// Mitsubishi GX Works2 project: 모터실린더완성2   PLC: Q02/Q02H

PROGRAM MAIN
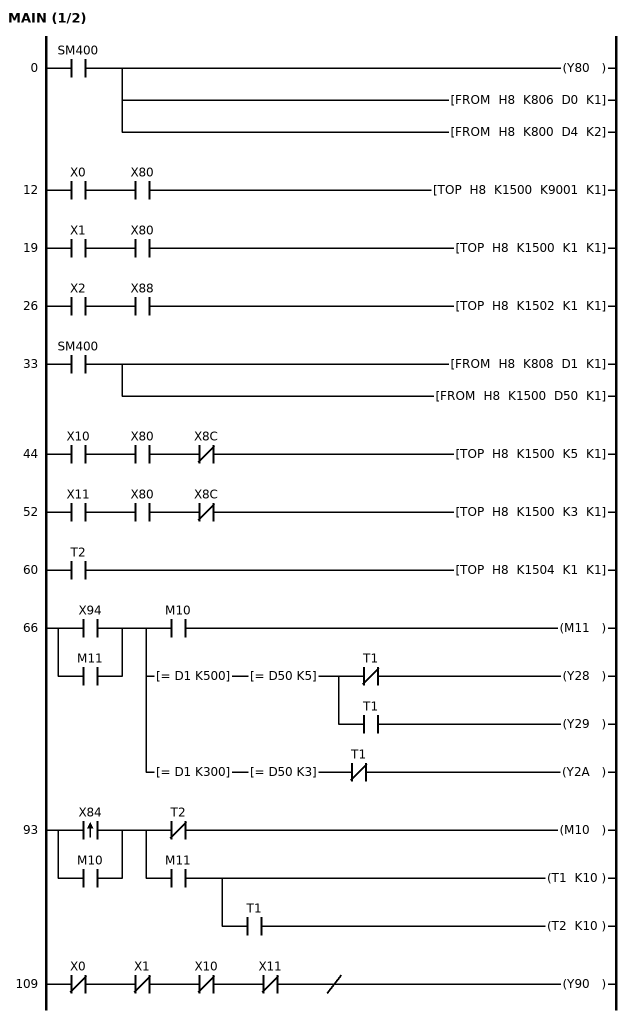
0     LD      SM400
      OUT     Y80
      FROM    H8 K806 D0 K1
      FROM    H8 K800 D4 K2
12    LD      X0
      AND     X80
      TOP     H8 K1500 K9001 K1
19    LD      X1
      AND     X80
      TOP     H8 K1500 K1 K1
26    LD      X2
      AND     X88
      TOP     H8 K1502 K1 K1
33    LD      SM400
      FROM    H8 K808 D1 K1
      FROM    H8 K1500 D50 K1
44    LD      X10
      AND     X80
      ANI     X8C
      TOP     H8 K1500 K5 K1
52    LD      X11
      AND     X80
      ANI     X8C
      TOP     H8 K1500 K3 K1
60    LD      T2
      TOP     H8 K1504 K1 K1
66    LD      X94
      OR      M11
      MPS
      AND     M10
      OUT     M11
      MRD
      AND=    D1 K500
      AND=    D50 K5
      MPS
      ANI     T1
      OUT     Y28
      MPP
      AND     T1
      OUT     Y29
      MPP
      AND=    D1 K300
      AND=    D50 K3
      ANI     T1
      OUT     Y2A
93    LDP     X84
      OR      M10
      MPS
      ANI     T2
      OUT     M10
      MPP
      AND     M11
      OUT     T1 K10
      AND     T1
      OUT     T2 K10
109   LDI     X0
      ANI     X1
      ANI     X10
      ANI     X11
      INV
      OUT     Y90
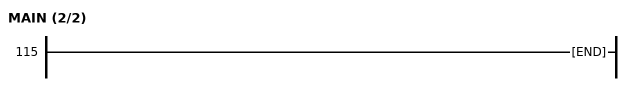
115   END
END_PROGRAM
